PROGRAM AnalogConversion
VAR
	i					: INT := 1; //charger 1-6
	m					: INT := 12; //numb of thermo
	
	ChargerV_UpRange	: REAL := 5;
	ChargerV_LoRange	: REAL := 0;
END_VAR

//MCP 

//AI
FOR i := 1 TO m BY 1 DO
	//exclude value when switch is off
	IF HMI_DB.ThermalCouple[i].IncludeSW = TRUE THEN 	
		MCP_IO.ThermalCouple[i].TemperatureFB:= INT_TO_REAL(MCP_IO.ThermalCouple[i].Temperature_raw)/10;
		//voltage
		//MCP_IO.ThermalCouple[i].Temperature_norm := Norm_x (raw_input := INT_TO_REAL (MCP_IO.ThermalCouple[i].Temperature_raw),
		//												x_max := 32767,
		//												x_min := 0);

		//MCP_IO.ThermalCouple[i].TemperatureFB := (HMI_DB.ThermalCoupleUpperRange - HMI_DB.ThermalCoupleLowerRange) * ADC_10V(
		//																					normal_input := MCP_IO.ThermalCouple[i].Temperature_norm,
		//																					x_max := 75,
		//																					x_min := -75);
	ELSIF HMI_DB.ThermalCouple[i].IncludeSW = FALSE THEN
		MCP_IO.ThermalCouple[i].TemperatureFB := 0;		
	END_IF;
END_FOR;



//Analog Output


// limit for the input 
IF HMI_DB.TemperatureSP > 100 THEN 
	//set limits of temperature input
	HMI_DB.TemperatureSP := 100; //limit at 100C
	ELSIF HMI_DB.TemperatureSP < 0 THEN 
		HMI_DB.TemperatureSP := 0;
END_IF; 

//hmi temperature setpoint input 
MCP_IO.TemperatureSP := HMI_DB.TemperatureSP;
		
//prepare output signal for 5V chargers.
//converting temperature sp 
MCP_IO.TemperatureSP_norm := Norm_x (raw_input := MCP_IO.TemperatureSP,
										x_max := HMI_DB.ThermalCoupleUpperRange, //1372 C
										x_min := HMI_DB.ThermalCoupleLowerRange); //-270 C

MCP_IO.TemperatureSP_raw := ADC_5V (normal_input := MCP_IO.TemperatureSP_norm,
												x_max := ChargerV_UpRange,
												x_min := ChargerV_LoRange);
												
												
//convert temp sp to range of 5V	- temperature sp raw -> PID to 5V

//	
MCP_IO.ChargerSP_norm := Norm_x (raw_input := MCP_IO.ChargerSP, 
									x_max := 32767,
									x_min := 0);	

//need to scale the temperature to the voltage first beforethe output												
MCP_IO.ChargerSP_raw := AQ_5V (norm_input := MCP_IO.ChargerSP_norm, 
												x_max := ChargerV_UpRange,
												x_min := ChargerV_LoRange);
												


												
	//limite for output sigal (<= 5V)  this should not happen
	IF MCP_IO.ChargerSP_raw >= 32767 THEN 
		MCP_IO.ChargerSP_raw := 32767; 										
	END_IF;
	



//reset counter
//IF i > 8 THEN
IF i > m THEN
	i := 1;
END_IF;

END_PROGRAM

(* stored: Version 1.1.0.1, ProductVersion 3.1.4024.11
   POU AnalogConversion: Id {8ae23b5e-db41-4801-a4ef-8d4e513d812d}, SpecialFunc None *)
